PROGRAM MAIN
VAR
	RequestedFloor AT%I*:INT;
	CurrentFloor AT%I*:INT;
	Motor AT%I*:ST_Motor;
	
	//BT_FloorCall AT %Q*:ARRAY[1..3]	OF	BOOL;
	LS_Floor AT %Q*:ARRAY[1..3]	OF	ST_LevelSensors;
	state: INT;
	nextState: INT;
	Timer:TON;
	TransitionTime:TIME:=T#3S;
END_VAR

IF	CurrentFloor=0 	THEN
	CurrentFloor:=1;
END_IF
IF	CurrentFloor>3	THEN
	CurrentFloor:=3;
END_IF

IF	RequestedFloor=0	THEN
	RequestedFloor:=1;
END_IF



IF	CurrentFloor>RequestedFloor	THEN
	//move down
	IF	NOT(state>=21 AND state<=211)	THEN
		state:=21;
	END_IF
ELSIF	CurrentFloor < RequestedFloor	THEN
	//moveUp
	IF	NOT(state>=1 AND state<=11)	THEN
		state:=1;
	END_IF
ELSE
	//arrive on the level
	IF	NOT(state>=13	AND	state<=15)	THEN
		state:=12;		
	END_IF

END_IF

CASE	state OF
	1:
		LS_Floor[CurrentFloor].Mid:=FALSE;
		state:=state+1;
		Timer(IN:= FALSE );
	2:
		Timer(IN:= TRUE, PT:= T#500MS );
		IF	timer.Q	THEN
			state:=state+1;
		END_IF
	3:
		LS_Floor[CurrentFloor].High:=TRUE;
		state:=state+1;
		Timer(IN:= FALSE );
	4:
		Timer(IN:= TRUE, PT:= T#500MS );
		IF	timer.Q	THEN
			state:=state+1;
		END_IF
	5:
		LS_Floor[CurrentFloor].High:=FALSE;
		state:=state+1;
		Timer(IN:= FALSE );
	6:
		Timer(IN:= TRUE, PT:= TransitionTime );
		IF	timer.Q	THEN
			state:=state+1;
		END_IF
	7:
		LS_Floor[CurrentFloor+1].Low:=TRUE;
		state:=state+1;
		Timer(IN:= FALSE );
	8:
		Timer(IN:= TRUE, PT:= T#500MS );
		IF	timer.Q	THEN
			state:=state+1;
		END_IF
	9:
		LS_Floor[CurrentFloor].Low:=FALSE;
		state:=state+1;
		Timer(IN:= FALSE );
	10:
		Timer(IN:= TRUE, PT:= T#500MS );
		IF	timer.Q	THEN
			state:=state+1;
		END_IF
	11:
		LS_Floor[CurrentFloor].Mid:=TRUE;
		state:=1;
		Timer(IN:= FALSE );
END_CASE

CASE	state OF
	21:
		LS_Floor[CurrentFloor].Mid:=FALSE;
		state:=state+1;
		Timer(IN:= FALSE );
	22:
		Timer(IN:= TRUE, PT:= T#500MS );
		IF	timer.Q	THEN
			state:=state+1;
		END_IF
	23:
		LS_Floor[CurrentFloor].Low:=TRUE;
		state:=state+1;
		Timer(IN:= FALSE );
	24:
		Timer(IN:= TRUE, PT:= T#500MS );
		IF	timer.Q	THEN
			state:=state+1;
		END_IF
	25:
		LS_Floor[CurrentFloor].Low:=FALSE;
		state:=state+1;
		Timer(IN:= FALSE );
	26:
		Timer(IN:= TRUE, PT:= TransitionTime);
		IF	timer.Q	THEN
			state:=state+1;
		END_IF
	27:
		LS_Floor[CurrentFloor-1].High:=TRUE;
		state:=state+1;
		Timer(IN:= FALSE );
	28:
		Timer(IN:= TRUE, PT:= T#500MS );
		IF	timer.Q	THEN
			state:=state+1;
		END_IF
	29:
		LS_Floor[CurrentFloor].High:=FALSE;
		state:=state+210;
		Timer(IN:= FALSE );
	210:
		Timer(IN:= TRUE, PT:= T#500MS );
		IF	timer.Q	THEN
			state:=state+1;
		END_IF
	211:
		LS_Floor[CurrentFloor].Mid:=TRUE;
		state:=21;
		Timer(IN:= FALSE );
END_CASE

CASE	state OF
	12:
		Timer(IN:= TRUE, PT:= T#500MS );
		IF	timer.Q	THEN
			state:=state+1;
		END_IF
	13:
		LS_Floor[CurrentFloor].Low:=
		LS_Floor[CurrentFloor].High:=FALSE;
		state:=state+1;
		Timer(IN:= FALSE );
	14:
		Timer(IN:= TRUE, PT:= T#500MS );
		IF	timer.Q	THEN
			state:=state+1;
		END_IF
	15:
		LS_Floor[CurrentFloor].Mid:=TRUE;
		state:=12;
		Timer(IN:= FALSE );
END_CASE

END_PROGRAM

(* stored: Version 1.1.0.1, ProductVersion 3.1.4024.11
   POU MAIN: Id {ca104f89-1b60-4670-b34e-7abdaf68ebfc}, SpecialFunc None *)
